(* IEC 61131-3 sources: elnaProjects/ElpcLogic/PomarKc7Changed/FunctionBlocks (part 3) *)

(* ---- Распаковка команды ---- *)
_sunpackerCommand(command := StrSw.inCommand);
	cmd := _sunpackerCommand.cmd;
	source := _sunpackerCommand.source;

(* ---- Обработка команды ---- *)
IF cmd <> 0 AND lastCmd <> cmd and (((NOT StrSw.opcCommandsDisabled) AND source > 0) OR source = 0) then
	CASE BYTE_TO_INT(cmd) OF
	(*cmd_open*) 1 :
			IF  StrSw.ISVALIDREF_cmdOn THEN StrSw.CmdOn := TRUE;
				IF StrSw.ISVALIDREF_cmdOff THEN StrSw.CmdOff := FALSE; END_IF;
			ELSIF  StrSw.ISVALIDREF_cmdOff THEN StrSw.CmdOff := FALSE;  END_IF;
			errorCMDTimer(IN := false);
			_commandErrorTimer := true;
			StrSw.lastCmdIsOn := true;
	(*cmd_close*) 2 :
			IF StrSw.ISVALIDREF_cmdOff THEN StrSw.CmdOff := TRUE;
				IF StrSw.ISVALIDREF_cmdOn THEN StrSw.CmdOn := FALSE; END_IF;
			ELSIF StrSw.ISVALIDREF_cmdOn THEN StrSw.CmdOn := FALSE; END_IF;
			errorCMDTimer(IN := false);
			_commandErrorTimer := true;
			StrSw.lastCmdIsOn := false;
	(*cmd_reset*) 3 :    IF StrSw.ISVALIDREF_statOn OR StrSw.ISVALIDREF_statOff THEN
			StrSw.CmdOn := FALSE;
			StrSw.CmdOff := FALSE;
                              lastCmd := 0;
			_commandErrorTimer := false;
			StrSw.lastCmdIsOn := false;
                               END_IF;
	END_CASE;
	source_for_Status := source;
	cmd_for_Status := cmd;
	command_error_for_Status := 0;
END_IF;
lastCmd := cmd;

errorCMDTimer(In := _commandErrorTimer, PT :=T#10s);

(* ---- алгоритм  для команды ВКЛючить ---- *)
IF (StrSw.onStatus = _statusDualInput.STATUS_ON) and (StrSw.lastCmdIsOn) then
	IF StrSw.ISVALIDREF_cmdOn AND StrSw.ISVALIDREF_cmdOff then  StrSw.cmdOn := false; END_IF;

	 errorCMDTimer(In := false);
	 _commandErrorTimer := false;
	 cmd_for_Status := 0;
	 source_for_Status := 0;
END_IF;

(* ---- off ---- *)
IF (StrSw.onStatus = _statusDualInput.STATUS_OFF) and (NOT StrSw.lastCmdIsOn) then
	IF StrSw.ISVALIDREF_cmdOn AND StrSw.ISVALIDREF_cmdOff then  StrSw.cmdOff := false; END_IF;

	 errorCMDTimer(In := false);
	 _commandErrorTimer := false;
	 cmd_for_Status := 0;
	 source_for_Status := 0;
END_IF;

(* ---- ошибка исполнения команды ---- *)
if errorCMDTimer.Q and (cmd_for_Status <> 0) then
	command_error_for_Status :=  cmd_for_Status;
	_commandErrorTimer := false;
	StrSw.CmdOn := false;
	StrSw.CmdOff := false;
	lastCmd := 0;
end_if;

(* ---- сброс ошибки команды ---- *)
StrSw.CommandFault := command_error_for_Status <> 0;
_errorReset(IN := command_error_for_Status <> 0, PT := T#5S);
IF _errorReset.Q THEN
	cmd_for_Status := 0;
	source_for_Status := 0;
	command_error_for_Status := 0;
END_IF;

outputsSets(in := (StrSw.ISVALIDREF_cmdOn and StrSw.cmdOn ) OR (StrSw.ISVALIDREF_cmdOff and StrSw.cmdOff), PT := T#2S);
	IF NOT outputsSets.Q THEN
		StrSw.BreakCmdOn := inBreakCmdOn._inversed AND inBreakCmdOn.reliability AND StrSw.ISVALIDREF_inBreakCmdOn;
		StrSw.BreakCmdOff := inBreakCmdOff._inversed AND inBreakCmdOff.reliability AND StrSw.ISVALIDREF_inBreakCmdOff;
	END_IF;

cmdOn := StrSw.cmdOn;
cmdOff:= StrSw.cmdOff;

(* ---- формирование зашифрованного статуса для АРМа ---- *)
StrSw.status := shl(BYTE_TO_DWORD(source_for_Status), 29)
		OR shl(BYTE_TO_DWORD(cmd_for_Status), 26)
		OR shl(BYTE_TO_DWORD(command_error_for_Status), 23)
		OR shl(bool_to_DWORD(StrSw.sdvig), 22)
		OR shl(bool_to_DWORD(StrSw.OpcCommandsDisabled), 21)
                    OR shl(BOOL_TO_DWORD(StrSw.offKNA), 17)
                    OR shl(bool_to_DWORD(StrSw.lastCmdIsOn), 14)
                    OR shl(BOOL_TO_DWORD(StrSw.BreakCmdOff), 13)
		OR shl(BOOL_TO_DWORD(StrSw.BreakCmdOn), 12)
                    OR shl(BYTE_TO_DWORD(StrSw.basketStatus), 8)
		OR shl(BOOL_TO_DWORD(StrSw.Distance), 6)
		OR shl(BOOL_TO_DWORD(StrSw.Local), 5)
		OR shl(BOOL_TO_DWORD(StrSw.Ns), 4)
                	OR shl(BOOL_TO_DWORD(StrSw.Accident ),3)
		OR BYTE_TO_DWORD(StrSw.onStatus);

(* ---- fb_SectionSwitch_Init.st ---- *)
FUNCTION_BLOCK fb_SectionSwitch_Init

VAR_INPUT
	data_Ini : BOOL; (*Флаг необходимости инициализации параметров.*)
	ISVALIDREF_statOn : BOOL;
	ISVALIDREF_statOff : BOOL;
	ISVALIDREF_cmdOn : BOOL;
	ISVALIDREF_cmdOff : BOOL;
	ISVALIDREF_inBreakCmdOn : BOOL;
	ISVALIDREF_inBreakCmdOff : BOOL;
	ISVALIDREF_basketRolledIn : BOOL;
	ISVALIDREF_basketRolledOut : BOOL;
	ISVALIDREF_basketTest : BOOL;
END_VAR

VAR_IN_OUT
	str_Sw : struct_SectionSwitch; (*Дескриптор AI-канала.*)
END_VAR

VAR_OUTPUT
	Init : BOOL          := FALSE; (*Флаг успешно выполненной инициализации.*)
END_VAR

(*****            Функциональный блок переинициализации структуры  МВ          *****)

 Init := FALSE;

    IF data_Ini THEN                            (* Параметрам требуется переинициализация. *)
        str_Sw.ISVALIDREF_statOn                := ISVALIDREF_statOn;
        str_Sw.ISVALIDREF_statOff               := ISVALIDREF_statOff;
        str_Sw.ISVALIDREF_cmdOn                 := ISVALIDREF_cmdOn;
        str_Sw.ISVALIDREF_cmdOff                := ISVALIDREF_cmdOff;
        str_Sw.ISVALIDREF_inBreakCmdOn          := ISVALIDREF_inBreakCmdOn;
        str_Sw.ISVALIDREF_inBreakCmdOff         := ISVALIDREF_inBreakCmdOff;
        str_Sw.ISVALIDREF_basketRolledIn        := ISVALIDREF_basketRolledIn;
        str_Sw.ISVALIDREF_basketRolledOut       := ISVALIDREF_basketRolledOut;
        str_Sw.ISVALIDREF_basketTest            := ISVALIDREF_basketTest;
        data_Ini:=FALSE;
        Init := TRUE;
    END_IF;
IF Init THEN
        ISVALIDREF_statOn:= FALSE;
        ISVALIDREF_statOff:= FALSE;
        ISVALIDREF_cmdOn:= FALSE;
        ISVALIDREF_cmdOff:= FALSE;
        ISVALIDREF_inBreakCmdOn:= FALSE;
        ISVALIDREF_inBreakCmdOff:= FALSE;
        ISVALIDREF_basketRolledIn:= FALSE;
        ISVALIDREF_basketRolledOut:= FALSE;
        ISVALIDREF_basketTest:= FALSE;
END_IF;

(* ---- fb_singleOutput.st ---- *)
FUNCTION_BLOCK fb_singleOutput

VAR_IN_OUT
	signal : BOOL;
	str_SO : struct_singleOutput;
END_VAR

VAR
	pulseTimer : TON;
	resetCmdTimer : TON;
	TON_Command : TON;
	source : BYTE;
	cmd : BYTE;
	lastCmd : BYTE;
	source_for_Status : BYTE;
	cmd_for_Status : BYTE;
	command_error_for_Status : BYTE;
	pulseTimerPriznak : BOOL;
	resetCmdTimerPriznak : BOOL;
	_sunpackerCommand : fb_sunpackerCommand;
END_VAR

str_SO.OpcCommandsDisabled := str_SO.inOpcCommandsDisabled;

(* ---- Если управление с ВУ заблокировано, то передаем команду из алгоритма ---- *)
IF str_SO.inOpcCommandsDisabled THEN
	str_SO.inCommand := str_SO.inCommand_Alg;
ELSE (* иначе передаем команду с АРМа*)
	str_SO.inCommand := str_SO.inCommand_ARM;
END_IF;

(*Распаковка команды*)
_sunpackerCommand(command := str_SO.inCommand);
	cmd := _sunpackerCommand.cmd;
	source := _sunpackerCommand.source;

(*Обработка команды*)
IF cmd <> 0 AND lastCmd <> cmd and (((NOT str_SO.OpcCommandsDisabled) AND source > 0) OR source = 0) then
	CASE BYTE_TO_INT(cmd) OF
	(*cmd_on*) 1 :
			str_SO.Q := TRUE;
			pulseTimer(IN := FALSE);
			pulseTimerPriznak := FALSE;
			resetCmdTimer(IN := FALSE);
			resetCmdTimerPriznak := TRUE;
	(*cmd_off*) 2 :
			str_SO.Q := FALSE;
			pulseTimer(IN := FALSE);
			pulseTimerPriznak := FALSE;
			resetCmdTimer(IN := FALSE);
			resetCmdTimerPriznak := TRUE;
	(*cmd_pulse*) 3 :
			str_SO.Q := TRUE;
                              pulseTimer(IN := FALSE);
                              pulseTimerPriznak := TRUE;
			resetCmdTimer(IN := FALSE);
                              resetCmdTimerPriznak := FALSE;
	END_CASE;
	source_for_Status := source;
	cmd_for_Status := cmd;
	command_error_for_Status := 0;
END_IF;
lastCmd := cmd;

pulseTimer(IN := pulseTimerPriznak, PT := str_SO.wait_time);
pulseTimer();
IF pulseTimer.Q THEN
	pulseTimer(IN := FALSE);
	pulseTimerPriznak := FALSE;

	str_SO.Q := FALSE;

	source_for_Status := 0;
	cmd_for_Status := 0;
	command_error_for_Status := 0;
END_IF;

resetCmdTimer(IN := resetCmdTimerPriznak, PT := T#10S);
resetCmdTimer();
IF resetCmdTimer.Q THEN
	resetCmdTimer(IN := FALSE);
	resetCmdTimerPriznak := FALSE;

	source_for_Status := 0;
	cmd_for_Status := 0;
	command_error_for_Status := 0;
END_IF;

signal:= str_SO.Q;

(*TON_Command(IN:= (inCommand <> 0) AND (source = 0), PT:= T#2S);*)
    (*IF TON_Command.Q THEN*)
        (*inCommand := 0;*)
    (*END_IF;*)
str_SO.status :=                           shl(BYTE_TO_DWORD(source_for_Status), 29)
				OR shl(BYTE_TO_DWORD(cmd_for_Status), 26)
				OR shl(BYTE_TO_DWORD(command_error_for_Status), 23)
				OR shl(BOOL_TO_DWORD(str_SO.OpcCommandsDisabled), 21)
				OR BOOL_TO_DWORD(str_SO.Q);

(* ---- fb_singleOutput_Init.st ---- *)
FUNCTION_BLOCK fb_singleOutput_Init

VAR_INPUT
	data_Ini : BOOL; (*Флаг необходимости инициализации параметров.*)
	inOpcCommandsDisabled : BOOL;
	wait_time : TIME;
END_VAR

VAR_IN_OUT
	str_SO : struct_singleOutput; (*Дескриптор AI-канала.*)
END_VAR

VAR_OUTPUT
	Init : BOOL          := FALSE; (*Флаг успешно выполненной инициализации.*)
END_VAR

(*****            Функциональный блок переинициализации структуры  singleOutput          *****)

Init := FALSE;

    IF data_Ini THEN                            (* Параметрам требуется переинициализация. *)
        str_SO.inOpcCommandsDisabled    := inOpcCommandsDisabled;
        str_SO.wait_time                := wait_time;

         data_Ini:=FALSE;
        Init := TRUE;
    END_IF;
 IF Init THEN
        inOpcCommandsDisabled := FALSE;
        wait_time := T#0S;
   END_IF;

(* ---- fb_singleSignal.st ---- *)
FUNCTION_BLOCK fb_singleSignal

VAR_INPUT
	signal : TYPE_ReliableBit;
END_VAR

VAR_IN_OUT
	str_SS : struct_singleSignal;
END_VAR

VAR
	TimerOn : TON;
	TimerOff : TOF;
END_VAR

str_SS.reliability:=signal.reliability;

IF NOT str_SS.inverse THEN
TimerOn(IN:=(signal.value AND str_SS.reliability AND NOT str_SS.Disabled_Sig), PT:=str_SS.DelayOn);
ELSE
TimerOn(IN:=(signal._inversed AND str_SS.reliability AND NOT str_SS.Disabled_Sig), PT:=str_SS.DelayOn);
END_IF;

TimerOff(IN:=TimerOn.Q, PT:=str_SS.DelayOff);

str_SS.Q:=TimerOff.Q;

str_SS.status:= SHL(BOOL_TO_DWORD(NOT str_SS.reliability), 15)
	OR BOOL_TO_DWORD(str_SS.Q);

(* ---- fb_singleSignal_Init.st ---- *)
FUNCTION_BLOCK fb_singleSignal_Init

VAR_INPUT
	data_Ini : BOOL; (*Флаг необходимости инициализации параметров.*)
	inverse : BOOL;
	DelayOn : TIME;
	DelayOff : TIME;
END_VAR

VAR_IN_OUT
	str_SS : struct_singleSignal; (*Дескриптор AI-канала.*)
END_VAR

VAR_OUTPUT
	Init : BOOL          := FALSE; (*Флаг успешно выполненной инициализации.*)
END_VAR

(*****            Функциональный блок переинициализации структуры  singleSignal          *****)
Init := FALSE;

    IF data_Ini THEN                            (* Параметрам требуется переинициализация. *)
        str_SS.inverse                := inverse;
        str_SS.DelayOn                := DelayOn;
        str_SS.DelayOff               := DelayOff;

        data_Ini:=FALSE;
        Init := TRUE;
    END_IF;
 IF Init THEN
        inverse := FALSE;
        DelayOn := T#0S;
        DelayOff:= T#0S;
 END_IF;

(* ---- fb_sunpackerCommand.st ---- *)
FUNCTION_BLOCK fb_sunpackerCommand

VAR_INPUT
	command : WORD;
END_VAR

VAR_OUTPUT
	source : BYTE;
	parametr : BYTE;
	cmd : BYTE;
END_VAR

cmd := WORD_TO_BYTE(command and 16#7);
parametr := WORD_TO_BYTE(SHR((command and 16#1FF8), 3));
source := WORD_TO_BYTE(SHR(command, 13));

(* ---- fb_Switch.st ---- *)
FUNCTION_BLOCK fb_Switch

VAR_INPUT
	statOn : BOOL;
	statOff : BOOL;
	statOn_reliability : BOOL;
	statOff_reliability : BOOL;
END_VAR

VAR_IN_OUT
	StrSw : struct_Switch;
END_VAR

VAR_INPUT
	inNs : TYPE_ReliableBit;
	inAccident : TYPE_ReliableBit;
	inAuto : TYPE_ReliableBit;
	inManual : TYPE_ReliableBit;
	inLocal : TYPE_ReliableBit;
	inDistance : TYPE_ReliableBit;
	inErrorPowerOff : TYPE_ReliableBit;
	inErrorBlock : TYPE_ReliableBit;
	inBreakCmdOn : TYPE_ReliableBit;
	inBreakCmdOff : TYPE_ReliableBit;
END_VAR

VAR
	onInit : BOOL          := FALSE;
	_statOn : BOOL;
	_statOff : BOOL;
	lastOnStatus : BYTE;
	cmd : BYTE;
	source : BYTE;
	lastCmd : BYTE;
	source_for_Status : BYTE;
	cmd_for_Status : BYTE;
	command_error_for_Status : BYTE;
	_sunpackerCommand : fb_sunpackerCommand;
	_statusDualInput : TYPE_statusDualInput;
	_commandDualInput : TYPE_commandDualInput;
	_commandErrorTimer : BOOL;
	resetErrorTimer : BOOL;
	getSdvig : BOOL;
	_changWithoutCommand : BOOL;
	errorCMDTimer : TON;
	sdvigReset : TON;
	_errorReset : TON;
	outputsSets : TOF;
END_VAR

VAR_IN_OUT
	cmdOn : BOOL;
	cmdOff : BOOL;
END_VAR

IF NOT onInit THEN
IF StrSw.ISVALIDREF_cmdOn XOR StrSw.ISVALIDREF_cmdOff THEN
	IF 	StrSw.ISVALIDREF_cmdOn THEN
		lastCmd:= 2; (*baseCmdOff*)
	ELSE
		lastCmd:= 1; (*baseCmdOn*)
	END_IF;
END_IF;
onInit:=TRUE;
END_IF;

(* ---- Если управление с ВУ заблокировано, то в ИМ передаем команду из алгоритма ---- *)
IF StrSw.inOpcCommandsDisabled THEN
	StrSw.inCommand := StrSw.inCommand_Alg;
ELSE (* иначе передаем команду с АРМа*)
	StrSw.inCommand := StrSw.inCommand_ARM;
END_IF;

(* ---- Формирование состояния механизма ---- *)

IF (StrSw.ISVALIDREF_statOn) OR (StrSw.ISVALIDREF_statOff) THEN
	IF (StrSw.ISVALIDREF_statOn) AND (StrSw.ISVALIDREF_statOff) THEN
	StrSw.reliability:= statOn_reliability AND statOff_reliability;
		_statOn  := statOn;
		_statOff := statOff;
	ELSIF (StrSw.ISVALIDREF_statOn) THEN
                     StrSw.reliability:= statOn_reliability;
		_statOn  := statOn;
		_statOff := NOT statOn;
	ELSIF (StrSw.ISVALIDREF_statOff) THEN
		 StrSw.reliability:= statOff_reliability;
		_statOn  := NOT statOff;
		_statOff :=statOff;
	END_IF;

	IF StrSw.reliability THEN
		IF _statOn AND NOT _statOff 		THEN 	StrSw.onStatus := _statusDualInput.STATUS_ON;
		ELSIF _statOff AND NOT _statOn 	THEN 	StrSw.onStatus := _statusDualInput.Status_OFF;
		ELSIF NOT _statOn AND NOT _statOff 	THEN 	StrSw.onStatus := _statusDualInput.STATUS_TRANSITIONAL;
		ELSE					StrSw.onStatus := _statusDualInput.STATUS_ERROR;
                    END_IF;

	ELSE
		StrSw.onStatus := _statusDualInput.STATUS_NOTDEFINED;

	END_IF;
ELSE
	CASE BYTE_TO_INT(lastCmd) OF
		(*baseCmdOn*) 1: StrSw.onStatus  := _statusDualInput.STATUS_ON;
		(*baseCmdOff*) 2: StrSw.onStatus  := _statusDualInput.STATUS_OFF;

	ELSE
		 StrSw.onStatus := _statusDualInput.STATUS_NOTDEFINED;

	END_CASE;
END_IF;

StrSw.Accident := inAccident.value AND inAccident.reliability;
StrSw.Ns := inNs.value AND inNs.reliability;
StrSw.Auto := inAuto.value AND inAuto.reliability;
StrSw.Manual := inManual.value AND inManual.reliability;
StrSw.Local := inLocal.value AND inLocal.reliability;
StrSw.Distance := inDistance.value AND inDistance.reliability;
StrSw.ErrorPowerOff := inErrorPowerOff.value AND inErrorPowerOff.reliability;
StrSw.ErrorBlock := inErrorBlock.value AND inErrorBlock.reliability;
StrSw.OpcCommandsDisabled := StrSw.inOpcCommandsDisabled;

(* ---- Формирование признака сдвига ---- *)
getSdvig := FALSE;
IF (StrSw.ISVALIDREF_cmdOn OR StrSw.ISVALIDREF_cmdOff) AND NOT StrSw.Local THEN
	IF NOT (StrSw.CmdOn OR StrSw.CmdOff) THEN
                     IF (lastOnStatus <> StrSw.onStatus AND
		(StrSw.onStatus <> _statusDualInput.STATUS_NOTDEFINED AND
                     StrSw.onStatus <> _statusDualInput.STATUS_ERROR)     AND
		(lastOnStatus <> _statusDualInput.STATUS_NOTDEFINED   AND
                     lastOnStatus <> _statusDualInput.STATUS_ERROR))
                    THEN
			getSdvig   := TRUE;
		END_IF;
	END_IF;
END_IF;

IF getSdvig THEN StrSw.sdvig:= TRUE; END_IF;

sdvigReset(IN:=StrSw.sdvig, PT:=T#15S);

IF sdvigReset.Q THEN StrSw.sdvig:=FALSE; END_IF;

lastOnStatus := StrSw.onStatus;

(* ---- Распаковка команды ---- *)
_sunpackerCommand(command := StrSw.inCommand);
	cmd := _sunpackerCommand.cmd;
	source := _sunpackerCommand.source;

(* ---- Обработка команды ---- *)
IF cmd <> 0 AND lastCmd <> cmd and (((NOT StrSw.opcCommandsDisabled) AND source > 0) OR source = 0) then
	CASE BYTE_TO_INT(cmd) OF
	(*cmd_open*) 1 :
			IF  StrSw.ISVALIDREF_cmdOn THEN StrSw.CmdOn := TRUE;
				IF StrSw.ISVALIDREF_cmdOff THEN StrSw.CmdOff := FALSE; END_IF;
			ELSIF  StrSw.ISVALIDREF_cmdOff THEN StrSw.CmdOff := FALSE;  END_IF;
                              lastCmd := cmd;
			errorCMDTimer(IN := false);
			_commandErrorTimer := true;
			StrSw.lastCmdIsOn := true;
	(*cmd_close*) 2 :
			IF StrSw.ISVALIDREF_cmdOff THEN StrSw.CmdOff := TRUE;
				IF StrSw.ISVALIDREF_cmdOn THEN StrSw.CmdOn := FALSE; END_IF;
			ELSIF StrSw.ISVALIDREF_cmdOn THEN StrSw.CmdOn := FALSE; END_IF;
                              lastCmd := cmd;
			errorCMDTimer(IN := false);
			_commandErrorTimer := true;
			StrSw.lastCmdIsOn := false;
	(*cmd_reset*) 3 :    IF StrSw.ISVALIDREF_statOn OR StrSw.ISVALIDREF_statOff THEN
			StrSw.CmdOn := FALSE;
			StrSw.CmdOff := FALSE;
                              lastCmd :=0;
			_commandErrorTimer := false;
			StrSw.lastCmdIsOn := false;
                               END_IF;
	END_CASE;
	source_for_Status := source;
	cmd_for_Status := cmd;
	command_error_for_Status := 0;
END_IF;

errorCMDTimer(In := _commandErrorTimer, PT :=T#10s);

(* ---- алгоритм  для команды ВКЛючить ---- *)
IF (StrSw.onStatus = _statusDualInput.STATUS_ON) and StrSw.lastCmdIsOn then
	IF StrSw.ISVALIDREF_cmdOn AND StrSw.ISVALIDREF_cmdOff then  StrSw.cmdOn := false; END_IF;

	 errorCMDTimer(In := false);
	 _commandErrorTimer := false;
	 cmd_for_Status := 0;
	 source_for_Status := 0;
END_IF;

(* ---- off ---- *)
IF (StrSw.onStatus = _statusDualInput.STATUS_OFF) and (NOT StrSw.lastCmdIsOn) then
	IF StrSw.ISVALIDREF_cmdOn AND StrSw.ISVALIDREF_cmdOff then  StrSw.cmdOff := false; END_IF;

	 errorCMDTimer(In := false);
	 _commandErrorTimer := false;
	 cmd_for_Status := 0;
	 source_for_Status := 0;
END_IF;

(* ---- ошибка исполнения команды ---- *)
if errorCMDTimer.Q and (cmd_for_Status <> 0) then
	command_error_for_Status :=  cmd_for_Status;
	_commandErrorTimer := false;
	StrSw.CmdOn := false;
	StrSw.CmdOff := false;
	lastCmd := 0;
end_if;

(* ---- сброс ошибки команды ---- *)
StrSw.CommandFault := command_error_for_Status <> 0;
_errorReset(IN := command_error_for_Status <> 0, PT := T#5S);
IF _errorReset.Q THEN
	cmd_for_Status := 0;
	source_for_Status := 0;
	command_error_for_Status := 0;
END_IF;

outputsSets(in := (StrSw.ISVALIDREF_cmdOn and StrSw.cmdOn ) OR (StrSw.ISVALIDREF_cmdOff and StrSw.cmdOff), PT := T#2S);
	IF NOT outputsSets.Q THEN
		StrSw.BreakCmdOn := inBreakCmdOn._inversed AND
                    inBreakCmdOn.reliability AND StrSw.ISVALIDREF_inBreakCmdOn;

		StrSw.BreakCmdOff := inBreakCmdOff._inversed
                    AND inBreakCmdOff.reliability AND StrSw.ISVALIDREF_inBreakCmdOff;
	END_IF;

cmdOn := StrSw.cmdOn;
cmdOff:= StrSw.cmdOff;

(* ---- формирование зашифрованного статуса для АРМа ---- *)
StrSw.status := shl(BYTE_TO_DWORD(source_for_Status), 29)
		OR shl(BYTE_TO_DWORD(cmd_for_Status), 26)
		OR shl(BYTE_TO_DWORD(command_error_for_Status), 23)
		OR shl(bool_to_DWORD(StrSw.sdvig), 22)
		OR shl(bool_to_DWORD(StrSw.OpcCommandsDisabled), 21)
                    OR shl(bool_to_DWORD(StrSw.lastCmdIsOn), 14)
                    OR shl(BOOL_TO_DWORD(StrSw.BreakCmdOff), 13)
		OR shl(BOOL_TO_DWORD(StrSw.BreakCmdOn), 12)
		OR shl(BOOL_TO_DWORD(StrSw.ErrorBlock), 11)
		OR shl(BOOL_TO_DWORD(StrSw.ErrorPowerOff), 10)
		OR shl(BOOL_TO_DWORD(StrSw.Manual), 8)
		OR shl(BOOL_TO_DWORD(StrSw.Auto), 7)
		OR shl(BOOL_TO_DWORD(StrSw.Distance), 6)
		OR shl(BOOL_TO_DWORD(StrSw.Local), 5)
		OR shl(BOOL_TO_DWORD(StrSw.Ns), 4)
                	OR shl(BOOL_TO_DWORD(StrSw.Accident ),3)
		OR BYTE_TO_DWORD(StrSw.onStatus);

(* ---- fb_Switch_Init.st ---- *)
FUNCTION_BLOCK fb_Switch_Init

VAR_INPUT
	data_Ini : BOOL; (*Флаг необходимости инициализации параметров.*)
	ISVALIDREF_statOn : BOOL;
	ISVALIDREF_statOff : BOOL;
	ISVALIDREF_cmdOn : BOOL;
	ISVALIDREF_cmdOff : BOOL;
	ISVALIDREF_inBreakCmdOn : BOOL;
	ISVALIDREF_inBreakCmdOff : BOOL;
END_VAR

VAR_IN_OUT
	str_Sw : struct_Switch;
END_VAR

VAR_OUTPUT
	Init : BOOL          := FALSE; (*Флаг успешно выполненной инициализации.*)
END_VAR

(*****            Функциональный блок переинициализации структуры  Switch          *****)

 Init := FALSE;

    IF data_Ini THEN                            (* Параметрам требуется переинициализация. *)
        str_Sw.ISVALIDREF_statOn                := ISVALIDREF_statOn;
        str_Sw.ISVALIDREF_statOff               := ISVALIDREF_statOff;
        str_Sw.ISVALIDREF_cmdOn                 := ISVALIDREF_cmdOn;
        str_Sw.ISVALIDREF_cmdOff                := ISVALIDREF_cmdOff;
        str_Sw.ISVALIDREF_inBreakCmdOn          := ISVALIDREF_inBreakCmdOn;
        str_Sw.ISVALIDREF_inBreakCmdOff         := ISVALIDREF_inBreakCmdOff;
        data_Ini:=FALSE;
        Init := TRUE;
    END_IF;
IF Init THEN
        ISVALIDREF_statOn:= FALSE;
        ISVALIDREF_statOff:= FALSE;
        ISVALIDREF_cmdOn:= FALSE;
        ISVALIDREF_cmdOff:= FALSE;
        ISVALIDREF_inBreakCmdOn:= FALSE;
        ISVALIDREF_inBreakCmdOff:= FALSE;
END_IF;

(* ---- fb_TableValue_Max.st ---- *)
FUNCTION_BLOCK fb_TableValue_Max

VAR_INPUT
	parametr : REAL;
END_VAR

VAR
	_table : ARRAY [0..8] OF TYPE_TableRec;
END_VAR

VAR_INPUT
	inverse : BOOL          := FALSE;
END_VAR

VAR_IN_OUT
	actualValue : REAL;
END_VAR

VAR
	indexLess : INT          := -1;
	indexMore : INT          := -1;
	Vali : REAL;
	i : INT;
	moreDistance : REAL;
	lessDistance : REAL;
	onInit : BOOL;
	_prevParam : REAL          := 50.0;
END_VAR

VAR CONSTANT
	maxTableLength : INT          := 9;
END_VAR

IF NOT onInit THEN
_table[0].x:=-35.0;  _table[0].y:=320.0;
_table[1].x:=-25.0;  _table[1].y:=315.0;
_table[2].x:=-15.0;  _table[2].y:=310.0;
_table[3].x:= -5.0;  _table[3].y:=305.0;
_table[4].x:=  0.0;  _table[4].y:=300.0;
_table[5].x:=  5.0;  _table[5].y:=295.0;
_table[6].x:= 15.0;  _table[6].y:=290.0;
_table[7].x:= 25.0;  _table[7].y:=285.0;
_table[8].x:= 35.0;  _table[8].y:=280.0;

onInit:=TRUE;
END_IF;

IF parametr <> _prevParam THEN
indexLess:=-1;
indexMore:=-1;
lessDistance:=0.0;
moreDistance:=0.0;
FOR i:=0 TO maxTableLength-1 DO
	IF NOT inverse THEN
		Vali:=_table[i].x;
	ELSE
		Vali:=_table[i].y;
	END_IF;

	IF (Vali=parametr) THEN
		indexLess:=i;
		indexMore:=i;
	ELSIF ((Vali<parametr) AND ((lessDistance>parametr-Vali) OR (indexLess<0))) THEN
		indexLess:=i;
		lessDistance:=parametr-Vali;
	ELSIF ((Vali>parametr) AND ((moreDistance>Vali-parametr) OR (indexMore<0))) THEN
		indexMore:=i;
		moreDistance:=parametr-Vali;
	END_IF;
END_FOR;
(*
IF indexLess<0 THEN
	indexLess:=indexMore;
END_IF;

IF indexMore<0 THEN
	indexMore:=indexLess;
END_IF;
*)
  IF (_table[indexMore].x<>_table[indexLess].x) THEN
  actualValue:=_table[indexLess].y+((_table[indexMore].y-_table[indexLess].y)/(_table[indexMore].x-_table[indexLess].x))*(parametr-_table[indexLess].x);
  ELSE
  actualValue:=_table[indexLess].y;
  END_IF;
   _prevParam:= parametr;
END_IF;

(* ---- fb_TableValue_Min.st ---- *)
FUNCTION_BLOCK fb_TableValue_Min

VAR_INPUT
	parametr : REAL;
END_VAR

VAR
	_table : ARRAY [0..8] OF TYPE_TableRec;
END_VAR

VAR_INPUT
	inverse : BOOL          := FALSE;
END_VAR

VAR_IN_OUT
	actualValue : REAL;
END_VAR

VAR
	indexLess : INT          := -1;
	indexMore : INT          := -1;
	Vali : REAL;
	i : INT;
	moreDistance : REAL;
	lessDistance : REAL;
	onInit : BOOL;
	_prevParam : REAL          := 50.0;
END_VAR

VAR CONSTANT
	maxTableLength : INT          := 9;
END_VAR

IF NOT onInit THEN
_table[0].x:=-35.0;  _table[0].y:=130.0;
_table[1].x:=-25.0;  _table[1].y:=124.0;
_table[2].x:=-15.0;  _table[2].y:=118.0;
_table[3].x:= -5.0;  _table[3].y:=112.0;
_table[4].x:=  0.0;  _table[4].y:=108.0;
_table[5].x:=  5.0;  _table[5].y:=106.0;
_table[6].x:= 15.0;  _table[6].y:=104.0;
_table[7].x:= 25.0;  _table[7].y:=102.0;
_table[8].x:= 35.0;  _table[8].y:= 97.0;

onInit:=TRUE;
END_IF;

IF parametr <> _prevParam THEN
indexLess:=-1;
indexMore:=-1;
lessDistance:=0.0;
moreDistance:=0.0;
FOR i:=0 TO maxTableLength-1 DO
	IF NOT inverse THEN
		Vali:=_table[i].x;
	ELSE
		Vali:=_table[i].y;
	END_IF;

	IF (Vali=parametr) THEN
		indexLess:=i;
		indexMore:=i;
	ELSIF ((Vali<parametr) AND ((lessDistance>parametr-Vali) OR (indexLess<0))) THEN
		indexLess:=i;
		lessDistance:=parametr-Vali;
	ELSIF ((Vali>parametr) AND ((moreDistance>Vali-parametr) OR (indexMore<0))) THEN
		indexMore:=i;
		moreDistance:=parametr-Vali;
	END_IF;
END_FOR;
(*
IF indexLess<0 THEN
	indexLess:=indexMore;
END_IF;

IF indexMore<0 THEN
	indexMore:=indexLess;
END_IF;
*)
  IF (_table[indexMore].x<>_table[indexLess].x) THEN
  actualValue:=_table[indexLess].y+((_table[indexMore].y-_table[indexLess].y)/(_table[indexMore].x-_table[indexLess].x))*(parametr-_table[indexLess].x);
  ELSE
  actualValue:=_table[indexLess].y;
  END_IF;
   _prevParam:= parametr;
END_IF;

(* ---- fb_Timings.st ---- *)
FUNCTION_BLOCK fb_Timings

VAR_EXTERNAL CONSTANT
	req_Cycle : REAL;
END_VAR

VAR_EXTERNAL
	gF_T_100mSec : BOOL;
	gT_1Sec : BOOL;
	gF_T_1Sec : BOOL;
	gT_1Min : BOOL;
	gR_T_1Min : BOOL;
	gF_T_1Min : BOOL;
	del_T : REAL;
	cur_Cycle : REAL;
END_VAR

VAR
	Tmr_100_ms : REAL; (*Таймер меток времени 100 мс .*)
END_VAR

VAR_EXTERNAL
	T_1SEC : REAL;
END_VAR

VAR
	Tmr_1_s : REAL; (*Таймер меток времени 1 с .*)
	Tmr_1_min : REAL; (*Таймер меток времени 1 мин .*)
END_VAR

(* Обработка времени. *)
Tmr_100_ms := Tmr_100_ms + cur_Cycle;
gF_T_100mSec := FALSE;
IF Tmr_100_ms >= 0.1 THEN Tmr_100_ms := 0.0; gF_T_100mSec := TRUE; END_IF;

Tmr_1_s := Tmr_1_s + cur_Cycle;
gF_T_1Sec := FALSE;
IF Tmr_1_s >= 1.0 THEN Tmr_1_s := 0.0; gF_T_1Sec := TRUE; END_IF;

T_1SEC := T_1SEC + cur_Cycle;
gT_1Sec := FALSE;
IF T_1SEC >= 2.0 THEN T_1SEC := 0.0;
  ELSIF T_1SEC >= 1.0 THEN gT_1Sec := TRUE; END_IF;

IF Tmr_1_min > 60.0 THEN
    Tmr_1_min := 0.0; gF_T_1Min := gT_1Min; gT_1Min := NOT gT_1Min; gR_T_1Min := gT_1Min;
  ELSE
    Tmr_1_min := Tmr_1_min + cur_Cycle; gR_T_1Min := FALSE; gF_T_1Min := FALSE;
END_IF;
del_T:= cur_Cycle;

(* ---- fb_vibegPNSAlg.st ---- *)
FUNCTION_BLOCK fb_vibegPNSAlg

VAR_IN_OUT
	StrAlg : struct_Alg;
END_VAR

VAR
	autoPnsOff : struct_PhaseAlgoritm;
	waitVibeg : struct_PhaseAlgoritm;
	pnsOff : struct_PhaseAlgoritm;
	vibegEnd : struct_PhaseAlgoritm;
END_VAR

VAR_IN_OUT
	algContinue : struct_Question;
END_VAR

VAR
	fb_autoPnsOff : fb_ph_algoritm;
	fb_waitVibeg : fb_ph_Timer;
	fb_algContinue : fb_Question;
	fb_pnsOff : fb_ph_Switch;
	fb_vibegEnd : fb_ph_CustomPhase;
	_sunpackerCommand : fb_sunpackerCommand;
	_statusAi : TYPE_StatusAi;
	_Answers : TYPE_Answers;
	_statusDualInput : TYPE_statusDualInput;
	_DualStateImAction : TYPE_DualStateImAction;
	_PhaseAlgoritmAction : TYPE_PhaseAlgoritmAction;
	source : BYTE;
	cmd : BYTE;
	lastCmd : BYTE;
	source_for_Status : BYTE;
	cmd_for_Status : BYTE;
	command_error_for_Status : BYTE;
	resetCmdTimer : TON;
	resetCmdTimerPriznak : BOOL;
	onInit : BOOL;
	waitReset : TON;
END_VAR

VAR_EXTERNAL
	IM : ImConfig;
	algoritms : AlgoritmsConfig;
	ai : AiConfig;
	protections : ProtectionsConfig;
	AlgTimers : struct_AlgTimers;
END_VAR

IF NOT onInit THEN
 fb_autoPnsOff(phaseNumber:=0, act:=_reset, waitCompletion:=FALSE);
  fb_waitVibeg(phaseNumber:=1, delay:=T#300S);
     algContinue.AnswerVariants:=_Answers.ANS_YES;
     fb_pnsOff(phaseNumber:=2, act:=_off);
   fb_vibegEnd(phaseNumber:=14);
onInit:=TRUE;
END_IF;

 fb_autoPnsOff(StrPh:=autoPnsOff, alg:=algoritms.autoPns);
  fb_waitVibeg(StrPh:=waitVibeg, timer:=AlgTimers.vibegPNS_Timer);
fb_algContinue(StrQ:=algContinue);
     fb_pnsOff(StrPh:=pnsOff, Im:=IM.pns);
   fb_vibegEnd(StrPh:=vibegEnd);

IF StrAlg.isRuning THEN

StrAlg.hasError := autoPnsOff.error OR pnsOff.error;

    IF IM.pns.onStatus = _statusDualInput.STATUS_ON AND NOT vibegEnd.top THEN

	runPhase(vibegEnd);
          runPhase(waitVibeg);
          askQuestion(algContinue);

    END_IF;

    IF waitVibeg.top OR (algContinue.answer = _Answers.ANS_YES) THEN
	vibegEnd.top:=TRUE;
	resetPhase(waitVibeg);
          resetQuestion(algContinue);

          resetAiProtection(protections.Os_sdvig_nagnetatelja_minus);
          (*resetDiProtection(protections.Vibro_skorost_OP_shesterni_RED_T6);*)

	(*IM.SingleSignals.P_oil_low.Disabled_Sig:=TRUE;*)
	ai.Pmasla_posle_GNS.Disabled_LA:=TRUE;
          ai.Pmasla_posle_GNS.Disabled_LW:=TRUE;
          ai.Pmasla_posle_NU.Disabled_LW:=TRUE;
	runPhase(pnsOff);
    END_IF;

    StrAlg.isEnded:=pnsOff.top;

END_IF;

StrAlg.CanRun := StrAlg.inCanRun;
StrAlg.OpcCommandsDisabled := StrAlg.inOpcCommandsDisabled;

(* ---- Если управление с ВУ заблокировано, то  передаем команду из алгоритма ---- *)
IF StrAlg.inOpcCommandsDisabled THEN
	StrAlg.inCommand := StrAlg.inCommand_Alg;
ELSE (* иначе передаем команду с АРМа*)
	StrAlg.inCommand := StrAlg.inCommand_ARM;
END_IF;

_sunpackerCommand(command := StrAlg.inCommand);
	source := _sunpackerCommand.source;
	cmd := _sunpackerCommand.cmd;

IF cmd <> 0 AND lastCmd <> cmd AND (((NOT StrAlg.opcCommandsDisabled) AND source > 0) OR source = 0) then
	CASE BYTE_TO_INT(cmd) OF
		(*cmdRun*) 1: 	IF (StrAlg.CanRun) THEN
					StrAlg.isRuning := TRUE;
					StrAlg.isEnded := FALSE;
					StrAlg.hasError := FALSE;
					(*****************       OnRun       *****************)
                                                  runPhase(autoPnsOff);

					cmd_for_Status := cmd;
					source_for_Status := source;
					command_error_for_Status := 0;
				ELSE
					StrAlg.isRuning := FALSE;
					StrAlg.isEnded := FALSE;
					StrAlg.hasError 	:= FALSE;

					cmd_for_Status := 0;
					source_for_Status := source;
					command_error_for_Status := cmd;
				END_IF;
		(*cmdReset*) 2: 	StrAlg.isRuning := FALSE;
				StrAlg.isEnded := FALSE;
				StrAlg.hasError 	:= FALSE;

                                         (*****************       OnReset       *****************)
                                       waitReset(IN:=FALSE);
                                       resetPhase(autoPnsOff);
                                       resetPhase(waitVibeg);
                                       resetPhase(vibegEnd);
                                       resetPhase(pnsOff);
                                       resetQuestion(algContinue);

				cmd_for_Status := cmd;
				source_for_Status := source;
				command_error_for_Status := 0;
	END_CASE;
	resetCmdTimer(IN := false);
	resetCmdTimerPriznak := TRUE;
END_IF;
lastCmd := cmd;

resetCmdTimer(IN := resetCmdTimerPriznak, PT := T#5S);
IF resetCmdTimer.Q THEN
	resetCmdTimerPriznak := FALSE;
	source_for_Status := 0;
	cmd_for_Status := 0;
	command_error_for_Status := 0;
END_IF;

StrAlg.Start:= autoPnsOff.startStatus
            OR waitVibeg.startStatus
            OR pnsOff.startStatus
            OR vibegEnd.startStatus;

StrAlg.Error:= autoPnsOff.errorStatus
            OR waitVibeg.errorStatus
            OR pnsOff.errorStatus
            OR vibegEnd.errorStatus;

StrAlg.Top:=   autoPnsOff.topStatus
            OR waitVibeg.topStatus
            OR pnsOff.topStatus
            OR vibegEnd.topStatus;

(*TODO: TYPE PROGRAM CODE HERE*)
StrAlg.status :=  SHL(BYTE_TO_DWORD(source_for_Status), 29)
			OR SHL(BYTE_TO_DWORD(cmd_for_Status), 26)
			OR SHL(BYTE_TO_DWORD(command_error_for_Status), 23)
			OR SHL(BOOL_TO_DWORD(StrAlg.OpcCommandsDisabled ), 21)
			OR SHL(BOOL_TO_DWORD(StrAlg.hasError),4)
			OR SHL(BOOL_TO_DWORD(StrAlg.CanRun),2)
			OR SHL(BOOL_TO_DWORD(StrAlg.isEnded),1)
			OR BOOL_TO_DWORD(StrAlg.isRuning);

(* ---- fb_ZapasAlg.st ---- *)
FUNCTION_BLOCK fb_ZapasAlg

VAR_INPUT
	Q_actual : struct_AI;
END_VAR

VAR_IN_OUT
	StrAi : struct_AI;
END_VAR

VAR_INPUT
	Q_min : LREAL;
	Q_max : LREAL;
END_VAR

VAR
	_statusAi : TYPE_StatusAi;
END_VAR

IF (Q_actual.interval < _statusAi.normal) THEN
	StrAi.interval := _statusAi.NOTRELIABLE;
          strAI.status := 	SHL(BOOL_TO_DWORD(strAI.OpcCommandsDisabled ), 21)
		OR BYTE_TO_DWORD(strAI.interval);
	RETURN;
END_IF;

IF (Q_actual.value <10.0) THEN
	StrAi.interval := _statusAi.normal;
	StrAi.value:= 100.0;
          strAI.status := 	SHL(BOOL_TO_DWORD(strAI.OpcCommandsDisabled ), 21)
		OR BYTE_TO_DWORD(strAI.interval);
	RETURN;
END_IF;

strAI.opcCommandsDisabled := strAI.inopcCommandsDisabled ;
StrAi.interval:= _statusAi.normal;

StrAi.value:= ((Q_actual.value - Q_min)/(Q_max-Q_min))*100.0;

strAI.status := 	SHL(BOOL_TO_DWORD(strAI.OpcCommandsDisabled ), 21) (* Управление в ВУ заблокировано *)
		OR BYTE_TO_DWORD(strAI.interval);	              (* интервал *)

(* ---- fillingAlg.st ---- *)
FUNCTION_BLOCK fillingAlg

VAR_IN_OUT
	StrAlg : struct_Alg;
END_VAR

VAR
	BreakPuskTimer : struct_PhaseAlgoritm;
	kran3bOpen : struct_PhaseAlgoritm;
	kran4Open : struct_PhaseAlgoritm;
	waitAfterKran4 : struct_PhaseAlgoritm;
	kran5Close : struct_PhaseAlgoritm;
	didPKran1 : struct_PhaseAlgoritm;
	kran1Open : struct_PhaseAlgoritm;
	kran2Open : struct_PhaseAlgoritm;
	kran3bClose : struct_PhaseAlgoritm;
	kran4Close : struct_PhaseAlgoritm;
	RunProtection_kr1 : struct_PhaseAlgoritm;
	RunProtection_kr2 : struct_PhaseAlgoritm;
	waitAfterKran5 : struct_PhaseAlgoritm;
	testUnsuccessfulFilling : struct_PhaseAlgoritm;
	fb_BreakPuskTimer : fb_ph_Timer;
	fb_kran3bOpen : fb_ph_Kran;
	fb_kran4Open : fb_ph_Kran;
	fb_waitAfterKran4 : fb_ph_Timer;
	fb_kran5Close : fb_ph_Kran;
	fb_didPKran1 : fb_ph_CustomPhase;
	fb_kran1Open : fb_ph_Kran;
	fb_kran2Open : fb_ph_Kran;
	fb_kran3bClose : fb_ph_Kran;
	fb_kran4Close : fb_ph_Kran;
	fb_RunProtection_kr1 : fb_ph_DIprotection;
	fb_RunProtection_kr2 : fb_ph_DIprotection;
	fb_waitAfterKran5 : fb_ph_Timer;
	fb_testUnsuccessfulFilling : fb_ph_CustomPhase;
	_sunpackerCommand : fb_sunpackerCommand;
	_DualStateImAction : TYPE_DualStateImAction;
	_PhaseAlgoritmAction : TYPE_PhaseAlgoritmAction;
	source : BYTE;
	cmd : BYTE;
	lastCmd : BYTE;
	source_for_Status : BYTE;
	cmd_for_Status : BYTE;
	command_error_for_Status : BYTE;
	resetCmdTimer : TON;
	resetCmdTimerPriznak : BOOL;
	onInit : BOOL;
	waitReset : TON;
END_VAR

VAR_EXTERNAL
	IM : ImConfig;
	ai : AiConfig;
	protections : ProtectionsConfig;
	AlgTimers : struct_AlgTimers;
	algoritms : AlgoritmsConfig;
END_VAR

IF NOT onInit THEN

         fb_BreakPuskTimer(phaseNumber:=0, delay:=T#240S);
             fb_kran3bOpen(phaseNumber:=1, act:=_on);
              fb_kran4Open(phaseNumber:=2, act:=_on);
         fb_waitAfterKran4(phaseNumber:=3, delay:=T#10S);
             fb_kran5Close(phaseNumber:=4, act:=_off);
              fb_didPKran1(phaseNumber:=5);
              fb_kran1Open(phaseNumber:=7, act:=_on);
              fb_kran2Open(phaseNumber:=8, act:=_on);
            fb_kran3bClose(phaseNumber:=9, act:=_off);
             fb_kran4Close(phaseNumber:=10, act:=_off);
      fb_RunProtection_kr1(phaseNumber:=11, act:=_run);
      fb_RunProtection_kr2(phaseNumber:=12, act:=_run);
         fb_waitAfterKran5(phaseNumber:=13, delay:=T#60S);
fb_testUnsuccessfulFilling(phaseNumber:=17);

onInit:=TRUE;
END_IF;

         fb_BreakPuskTimer(StrPh:=BreakPuskTimer, timer:=AlgTimers.filling_BreakPuskTimer);
             fb_kran3bOpen(StrPh:=kran3bOpen, Im:=Im.kran3b);
              fb_kran4Open(StrPh:=kran4Open, Im:=Im.kran4);
         fb_waitAfterKran4(StrPh:=waitAfterKran4, timer:=AlgTimers.filling_waitAfterKran4);
             fb_kran5Close(StrPh:=kran5Close, Im:=Im.kran5);
              fb_didPKran1(StrPh:=didPKran1);
              fb_kran1Open(StrPh:=kran1Open, Im:=Im.kran1);
              fb_kran2Open(StrPh:=kran2Open, Im:=Im.kran2);
            fb_kran3bClose(StrPh:=kran3bClose, Im:=Im.kran3b);
             fb_kran4Close(StrPh:=kran4Close, Im:=Im.kran4);
      fb_RunProtection_kr1(StrPh:=RunProtection_kr1 , StrDiP:=protections.Reg_vozb_off);
      fb_RunProtection_kr2(StrPh:=RunProtection_kr2 , StrDiP:=protections.Fail_chastotnii_pusk);
         fb_waitAfterKran5(StrPh:=waitAfterKran5, timer:=AlgTimers.filling_waitAfterKran5);
fb_testUnsuccessfulFilling(StrPh:=testUnsuccessfulFilling);

StrAlg.CanRun := StrAlg.inCanRun;
StrAlg.OpcCommandsDisabled := StrAlg.inOpcCommandsDisabled;

IF StrAlg.isRuning THEN

    StrAlg.hasError := kran3bOpen.error OR kran4Open.error OR kran5Close.error OR kran5Close.error
    OR kran1Open.error OR kran2Open.error OR kran3bClose.error OR kran4Close.error OR testUnsuccessfulFilling.error;

    IF kran4Open.top THEN
        runPhase(waitAfterKran4);
    END_IF;

    IF waitAfterKran4.top THEN
        runPhase(kran5Close);
    END_IF;

    IF kran3bOpen.top AND kran5Close.top THEN
       runPhase(waitAfterKran5);
       runPhase(didPKran1);
    END_IF;

    (*IF didPKran1.start AND NOT didPKran1.top THEN
    didPKran1.top:= im.singleSignals.dP_gazgaz_Kran1.Q;
    END_IF;*)

    IF waitAfterKran5.top AND didPKran1.top THEN
          runPhase(kran1Open);
	runPhase(kran2Open);
    END_IF;

    IF kran1Open.top AND kran2Open.top THEN
          runPhase(kran4Close);
	runPhase(kran3bClose);
    END_IF;

    IF kran4Close.top AND kran3bClose.top THEN

          runPhase(RunProtection_kr1);
          runPhase(RunProtection_kr2);

          (*runAiProtection(protections.Pgaza_na_vhode_nagnetatelia);
          runAiProtection(protections.Pgaza_na_vhode_nagnetatelia);
          runAiProtection(protections.Pgaza_na_vyhode_nagnetatelia);
          runAiProtection(protections.dPmaslo_gaz);
          runAiProtection(protections.Pmaslo_sm_nizkoe);
          runAiProtection(protections.Pmaslo_sm_vysokoe);*)

    END_IF;

    IF BreakPuskTimer.top AND NOT (RunProtection_kr1.top AND RunProtection_kr2.top ) THEN
	testUnsuccessfulFilling.error:=TRUE;
    END_IF;

    IF RunProtection_kr1.top AND RunProtection_kr2.top THEN
          resetPhase(BreakPuskTimer);
	waitReset(IN:=TRUE, PT:= T#2S);
    END_IF;

    IF waitReset.Q AND NOT (algoritms.Apusk.isRuning OR algoritms.SemiAutoPusk.isRuning) THEN
	resetIfRunning(StrAlg);
    END_IF;

    StrAlg.isEnded:= RunProtection_kr1.top AND RunProtection_kr2.top;
END_IF;

StrAlg.CanRun := StrAlg.inCanRun;
StrAlg.OpcCommandsDisabled := StrAlg.inOpcCommandsDisabled;

(* ---- Если управление с ВУ заблокировано, то  передаем команду из алгоритма ---- *)
IF StrAlg.inOpcCommandsDisabled THEN
	StrAlg.inCommand := StrAlg.inCommand_Alg;
ELSE (* иначе передаем команду с АРМа*)
	StrAlg.inCommand := StrAlg.inCommand_ARM;
END_IF;

_sunpackerCommand(command := StrAlg.inCommand);
	source := _sunpackerCommand.source;
	cmd := _sunpackerCommand.cmd;

IF cmd <> 0 AND lastCmd <> cmd AND (((NOT StrAlg.opcCommandsDisabled) AND source > 0) OR source = 0) then
	CASE BYTE_TO_INT(cmd) OF
		(*cmdRun*) 1: 	IF (StrAlg.CanRun) THEN
					StrAlg.isRuning := TRUE;
					StrAlg.isEnded := FALSE;
					StrAlg.hasError := FALSE;
					(*****************       OnRun       *****************)

                                                  runPhase(kran3bOpen);
                                                  runPhase(kran4Open);
                                                  runPhase(BreakPuskTimer);
                                                  runPhase(testUnsuccessfulFilling);

					cmd_for_Status := cmd;
					source_for_Status := source;
					command_error_for_Status := 0;
				ELSE
					StrAlg.isRuning := FALSE;
					StrAlg.isEnded := FALSE;
					StrAlg.hasError 	:= FALSE;

					cmd_for_Status := 0;
					source_for_Status := source;
					command_error_for_Status := cmd;
				END_IF;
		(*cmdReset*) 2: 	StrAlg.isRuning := FALSE;
				StrAlg.isEnded := FALSE;
				StrAlg.hasError 	:= FALSE;

                                         (*****************       OnReset       *****************)
                                        StrAlg.inCanRun:=FALSE;
                                        waitReset(IN:=FALSE);

                                        resetPhase(BreakPuskTimer);
                                        resetPhase(kran3bOpen);
                                        resetPhase(kran4Open);
                                        resetPhase(waitAfterKran4);
                                        resetPhase(kran5Close);
                                        resetPhase(didPKran1);
                                        resetPhase(kran1Open);
                                        resetPhase(kran2Open);
                                        resetPhase(kran3bClose);
                                        resetPhase(kran4Close);
	                              resetPhase(RunProtection_kr1);
                                        resetPhase(RunProtection_kr2);
                                        resetPhase(waitAfterKran5);
                                        resetPhase(testUnsuccessfulFilling);

				cmd_for_Status := cmd;
				source_for_Status := source;
				command_error_for_Status := 0;
	END_CASE;
	resetCmdTimer(IN := false);
	resetCmdTimerPriznak := TRUE;
END_IF;
lastCmd := cmd;

resetCmdTimer(IN := resetCmdTimerPriznak, PT := T#5S);
IF resetCmdTimer.Q THEN
	resetCmdTimerPriznak := FALSE;
	source_for_Status := 0;
	cmd_for_Status := 0;
	command_error_for_Status := 0;
END_IF;

StrAlg.Start:= BreakPuskTimer.startStatus
            OR kran3bOpen.startStatus
            OR kran4Open.startStatus
            OR waitAfterKran4.startStatus
            OR kran5Close.startStatus
            OR didPKran1.startStatus
            OR kran1Open.startStatus
            OR kran2Open.startStatus
            OR kran3bClose.startStatus
            OR kran4Close.startStatus
            OR RunProtection_kr1.startStatus
            OR RunProtection_kr2.startStatus
            OR waitAfterKran5.startStatus
            OR testUnsuccessfulFilling.startStatus;

StrAlg.Error:= BreakPuskTimer.errorStatus
            OR kran3bOpen.errorStatus
            OR kran4Open.errorStatus
            OR waitAfterKran4.errorStatus
            OR kran5Close.errorStatus
            OR didPKran1.errorStatus
            OR kran1Open.errorStatus
            OR kran2Open.errorStatus
            OR kran3bClose.errorStatus
            OR kran4Close.errorStatus
            OR RunProtection_kr1.errorStatus
            OR RunProtection_kr2.errorStatus
            OR waitAfterKran5.errorStatus
            OR testUnsuccessfulFilling.errorStatus;

StrAlg.Top:=   BreakPuskTimer.topStatus
            OR kran3bOpen.topStatus
            OR kran4Open.topStatus
            OR waitAfterKran4.topStatus
            OR kran5Close.topStatus
            OR didPKran1.topStatus
            OR kran1Open.topStatus
            OR kran2Open.topStatus
            OR kran3bClose.topStatus
            OR kran4Close.topStatus
            OR RunProtection_kr1.topStatus
            OR RunProtection_kr2.topStatus
            OR waitAfterKran5.topStatus
            OR testUnsuccessfulFilling.topStatus;

(*TODO: TYPE PROGRAM CODE HERE*)
StrAlg.status :=  SHL(BYTE_TO_DWORD(source_for_Status), 29)
			OR SHL(BYTE_TO_DWORD(cmd_for_Status), 26)
			OR SHL(BYTE_TO_DWORD(command_error_for_Status), 23)
			OR SHL(BOOL_TO_DWORD(StrAlg.OpcCommandsDisabled ), 21)
			OR SHL(BOOL_TO_DWORD(StrAlg.hasError),4)
			OR SHL(BOOL_TO_DWORD(StrAlg.CanRun),2)
			OR SHL(BOOL_TO_DWORD(StrAlg.isEnded),1)
			OR BOOL_TO_DWORD(StrAlg.isRuning);

(* ---- NOAlg.st ---- *)
FUNCTION_BLOCK NOAlg

VAR_IN_OUT
	StrAlg : struct_Alg;
END_VAR

VAR
	timer120 : struct_PhaseAlgoritm;
	kran6Open : struct_PhaseAlgoritm;
	pnsOn : struct_PhaseAlgoritm;
	kran4Close : struct_PhaseAlgoritm;
	kran3bOpen : struct_PhaseAlgoritm;
	mvOff : struct_PhaseAlgoritm;
	kran1Close : struct_PhaseAlgoritm;
	kran2Close : struct_PhaseAlgoritm;
	kran3Close : struct_PhaseAlgoritm;
	kran5Open : struct_PhaseAlgoritm;
	error_Krans : struct_PhaseAlgoritm;
	autoPnsOff : struct_PhaseAlgoritm;
	Pg_VhodLessThen300 : struct_PhaseAlgoritm;
	Pg_VyhodLessThen300 : struct_PhaseAlgoritm;
	nu1off : struct_PhaseAlgoritm;
	nu2off : struct_PhaseAlgoritm;
	AutoNU_Off : struct_PhaseAlgoritm;
	timer600 : struct_PhaseAlgoritm;
	pnsOff : struct_PhaseAlgoritm;
	Avom1Off : struct_PhaseAlgoritm;
	Avom2Off : struct_PhaseAlgoritm;
	Avom3Off : struct_PhaseAlgoritm;
	Avom4Off : struct_PhaseAlgoritm;
	autoAVOMOff : struct_PhaseAlgoritm;
	timer5 : struct_PhaseAlgoritm;
	klapan1 : struct_PhaseAlgoritm;
	klapan2 : struct_PhaseAlgoritm;
	nu_On : struct_PhaseAlgoritm;
	fb_timer120 : fb_ph_Timer;
	fb_kran6Open : fb_ph_Kran;
	fb_pnsOn : fb_ph_Switch;
	fb_kran4Close : fb_ph_Kran;
	fb_kran3bOpen : fb_ph_Kran;
	fb_mvOff : fb_ph_SectionSwitch;
	fb_kran1Close : fb_ph_Kran;
	fb_kran2Close : fb_ph_Kran;
	fb_kran3Close : fb_ph_Kran;
	fb_kran5Open : fb_ph_Kran;
	fb_error_Krans : fb_ph_CustomPhase;
	fb_autoPnsOff : fb_ph_algoritm;
	fb_Pg_VhodLessThen300 : fb_ph_CustomPhase;
	fb_Pg_VyhodLessThen300 : fb_ph_CustomPhase;
	fb_nu1Off : fb_ph_OilPump;
	fb_nu2Off : fb_ph_OilPump;
	fb_autoNuOff : fb_ph_algoritm;
	fb_timer600 : fb_ph_Timer;
	fb_pnsOff : fb_ph_Switch;
	fb_Avom1Off : fb_ph_Switch;
	fb_Avom2Off : fb_ph_Switch;
	fb_Avom3Off : fb_ph_Switch;
	fb_Avom4Off : fb_ph_Switch;
	fb_autoAVOMOff : fb_ph_algoritm;
	fb_timer5 : fb_ph_Timer;
	fb_klapan1 : fb_ph_CustomPhase;
	fb_klapan2 : fb_ph_CustomPhase;
	fb_nu_On : fb_ph_CustomPhase;
	_sunpackerCommand : fb_sunpackerCommand;
	_statusAi : TYPE_StatusAi;
	_Answers : TYPE_Answers;
	_statusDualInput : TYPE_statusDualInput;
	_commandDualInput : TYPE_commandDualInput;
	_DualStateImAction : TYPE_DualStateImAction;
	_PhaseAlgoritmAction : TYPE_PhaseAlgoritmAction;
	source : BYTE;
	cmd : BYTE;
	lastCmd : BYTE;
	source_for_Status : BYTE;
	cmd_for_Status : BYTE;
	command_error_for_Status : BYTE;
	resetCmdTimer : TON;
	resetCmdTimerPriznak : BOOL;
	onInit : BOOL;
	waitReset : TON;
END_VAR

VAR_EXTERNAL
	IM : ImConfig;
	algoritms : AlgoritmsConfig;
	ai : AiConfig;
	protections : ProtectionsConfig;
	ModeGpa : TYPE_ModeGpa;
	algManager : struct_AlgoritmsManager;
	AlgTimers : struct_AlgTimers;
END_VAR

VAR CONSTANT
	Ust_Pgaza : LREAL          := 0.3;
END_VAR

IF NOT onInit THEN
    fb_timer120(phaseNumber:=1, delay:=T#120S);
    fb_kran6Open(phaseNumber:=2, act:=_on);
    fb_kran4Close(phaseNumber:=3, act:=_off);
    fb_kran3bOpen(phaseNumber:=4, act:=_off);
    fb_mvOff(phaseNumber:=5, act:=_off);
    fb_kran1Close(phaseNumber:=6, act:=_off);
    fb_kran2Close(phaseNumber:=7, act:=_off);
    fb_kran3Close(phaseNumber:=8, act:=_off);
    fb_kran5Open(phaseNumber:=9, act:=_on);
    fb_error_Krans(phaseNumber:=10);
    fb_autoPnsOff(phaseNumber:=11, act:=_reset, waitCompletion:=FALSE);
    fb_pnsOn(phaseNumber:=12, act:=_on);
    fb_Pg_VhodLessThen300(phaseNumber:=13);
    fb_Pg_VyhodLessThen300(phaseNumber:=14);
    fb_nu1Off(phaseNumber:=15, act:=_off);
    fb_nu2Off(phaseNumber:=16, act:=_off);
    fb_autoNuOff(phaseNumber:=17, act:=_reset, waitCompletion:=FALSE);
    fb_timer600(phaseNumber:=18, delay:=T#600S);
    fb_pnsOff(phaseNumber:=19, act:=_off);
    fb_Avom1Off(phaseNumber:=20, act:=_off);
    fb_Avom2Off(phaseNumber:=21, act:=_off);
    fb_Avom3Off(phaseNumber:=22, act:=_off);
    fb_Avom4Off(phaseNumber:=23, act:=_off);
    fb_autoAVOMOff(phaseNumber:=24, act:=_reset, waitCompletion:=FALSE);
    fb_timer5(phaseNumber:=25, delay:=T#5S);
    fb_klapan1(phaseNumber:=26);
    fb_klapan2(phaseNumber:=27);
    fb_nu_On(phaseNumber:=28);

onInit:=TRUE;
END_IF;

fb_timer120(StrPh:=timer120, timer:=AlgTimers.No_wait120);
fb_kran6Open(StrPh:=kran6Open, Im:=Im.kran6);
fb_pnsOn(StrPh:=pnsOn, Im:=Im.pns);
fb_kran4Close(StrPh:=kran4Close, Im:=Im.kran4);
fb_kran3bOpen(StrPh:=kran3bOpen, Im:=Im.kran3b);
fb_mvOff(StrPh:=mvOff, Im:=Im.mv);
fb_kran1Close(StrPh:=kran1Close, Im:=Im.kran1);
fb_kran2Close(StrPh:=kran2Close, Im:=Im.Kran2);
fb_kran3Close(StrPh:=kran3Close, Im:=Im.Kran3);
fb_kran5Open(StrPh:=kran5Open, Im:=Im.Kran5);
fb_error_Krans(StrPh:=error_Krans);
fb_autoPnsOff(StrPh:=autoPnsOff, alg:=algoritms.autoPns);
fb_Pg_VhodLessThen300(StrPh:=Pg_VhodLessThen300);
fb_Pg_VyhodLessThen300(StrPh:=Pg_VyhodLessThen300);
fb_nu1Off(StrPh:=nu1off, Im:=Im.nu1);
fb_nu2Off(StrPh:=nu2off, Im:=Im.nu2);
fb_autoNuOff(StrPh:=AutoNU_Off, alg:=algoritms.autoNu);
fb_timer600(StrPh:=timer600, timer:=AlgTimers.No_wait600);
fb_pnsOff(StrPh:=pnsOff, Im:=Im.pns);
fb_Avom1Off(StrPh:=Avom1Off, Im:=Im.v1_Avom);
fb_Avom2Off(StrPh:=Avom2Off, Im:=Im.v2_Avom);
fb_Avom3Off(StrPh:=Avom3Off, Im:=Im.v3_Avom);
fb_Avom4Off(StrPh:=Avom4Off, Im:=Im.v4_Avom);
fb_autoAVOMOff(StrPh:=autoAVOMOff, alg:=algoritms.AutoAvom);
fb_timer5(StrPh:=timer5, timer:=AlgTimers.No_wait5);
fb_klapan1(StrPh:=klapan1);
fb_klapan2(StrPh:=klapan2);
fb_nu_On(StrPh:=nu_On);

StrAlg.CanRun := StrAlg.inCanRun;
StrAlg.OpcCommandsDisabled := StrAlg.inOpcCommandsDisabled;

IF StrAlg.isRuning THEN
    (* кран 6 не открыт - запуск таймера *)
    IF NOT kran6Open.top AND NOT timer120.top  THEN
	runPhase(timer120);
    ELSE
    (* счетчик отработал и кран 6 не открыт - ошибка *)
        IF timer120.top AND NOT kran6Open.top THEN
            error_Krans.error := TRUE;
        END_IF;
    END_IF;

    (* старт смазки кранов *)
    IF (*algoritms.F3.Smazka_1_2 OR *)IM.kran1.onStatus = _statusDualInput.STATUS_ON OR IM.kran1.onStatus = _statusDualInput.STATUS_TRANSITIONAL
	OR IM.kran2.onStatus = _statusDualInput.STATUS_ON OR IM.kran2.onStatus = _statusDualInput.STATUS_TRANSITIONAL  THEN
        IF (*(algoritms.F3.Smazka_1_2 OR *)IM.kran1.onStatus = _statusDualInput.STATUS_ON OR IM.kran1.onStatus = _statusDualInput.STATUS_TRANSITIONAL AND NOT klapan1.start AND NOT kran1Close.top THEN
            runPhase(klapan1);
        END_IF;
        IF (*(algoritms.F3.Smazka_1_2 OR *)IM.kran2.onStatus = _statusDualInput.STATUS_ON OR IM.kran2.onStatus = _statusDualInput.STATUS_TRANSITIONAL AND NOT klapan2.start AND NOT kran2Close.top THEN
            runPhase(klapan2);
        END_IF;
    (*algoritms.F3.Smazka_1_2:=FALSE;*)
    END_IF;

    (* открыть кран 6 кран 4 *)
    runPhase(kran6Open);
    runPhase(kran4Close);

    (*не понимаю
    IF kran4Close.top THEN
        ystavki.Block_kr4_alg.setValue (0);
    END_IF;*)

    (* кран 6 открыт *)
    IF kran6Open.top THEN
	runPhase(kran3bOpen);
	resetPhase(timer120);
	(*error_Krans.top := FALSE;
	error_Krans.error := FALSE;*)
	(*algoritms.S_Vibr.CanRun:=FALSE;
	algoritms.S_Vibr.reset (); net takogo alg*)
    END_IF;
    IF kran3bOpen.top AND NOT mvoff.start THEN
	resetDiProtection(protections.mvOff);
	resetDiProtection(protections.Off_avar_vikluchatel);
	resetDiProtection(protections.Reg_vozb_off);
	runPhase(mvOff);
    END_IF;

    IF mvOff.top (*AND NOT flag1*) THEN
        algoritms.AutoPns.inCanRun :=FALSE;
        (*algoritms.AutoPNS_Start.reset (); nichego ne ponimau
        algoritms.AutoPns.inCanRun :=FALSE;*)
        runPhase(autoPnsOff);
        runPhase(pnsOn);
        resetDiProtection(protections.Kran1_sdvig);
        resetDiProtection(protections.Kran2_sdvig);
        runPhase(kran1Close);
        runPhase(kran2Close);
        runPhase(kran3Close);
        runPhase(nu_On);

        (*тут запустить насосы уплотнения *)

        (*algoritms.autoNu.inCanRun:=FALSE;
        algoritms.autoNu_2.reset ();
        algoritms.autoNu_1.inCanRun:=TRUE;
        algoritms.autoNu_1.run ();
        flag1:=TRUE; что тут происходит?*)
    END_IF;
    IF ((IM.nu1.onStatus =_statusDualInput.STATUS_ON) OR (IM.nu2.onStatus =_statusDualInput.STATUS_ON)) AND nu_On.start AND NOT nu_On.top THEN
        nu_On.top:=TRUE;
    END_IF;

    (* выдача смазки *)
    IF klapan1.start AND kran1Close.top THEN
        (*IM.Kr1_Smazka.impulse(); не понимаю((((((((*)
        klapan1.top:=TRUE;
    END_IF;

    IF klapan2.start AND kran2Close.top THEN
	(*IM.Kr2_Smazka.impulse(); не понимаю *)
	klapan2.top:=TRUE;
    END_IF;

    (* кран 1 кран 2 кран 3 кран 4 закрыты - открыть кран 5 *)
    IF kran1Close.top AND kran2Close.top AND kran3Close.top AND kran4Close.top THEN
        runPhase(kran5Open);
        resetAiProtection(protections.Pgaza_na_vyhode_nagnetatelia);
    END_IF;

    IF kran5Open.top THEN
        runPhase(Pg_VhodLessThen300);
        runPhase(Pg_VyhodLessThen300);
    END_IF;

    IF Pg_VhodLessThen300.start AND NOT Pg_VhodLessThen300.top THEN
        IF (ai.Pgaza_na_vhode_nagnetatelia.interval>= _statusAi.NORMAL) AND (ai.Pgaza_na_vhode_nagnetatelia.value < 0.3) THEN
            Pg_VhodLessThen300.top:=TRUE;
        END_IF;
    END_IF;

    IF Pg_VyhodLessThen300.start AND NOT Pg_VyhodLessThen300.top THEN
        IF (ai.Pgaza_na_vyhode_nagnetatelia.interval>=_statusAi.NORMAL) AND (ai.Pgaza_na_vyhode_nagnetatelia.value < 0.3) THEN
            Pg_VyhodLessThen300.top:=TRUE;
        END_IF;
    END_IF;

    IF Pg_VhodLessThen300.top AND Pg_VyhodLessThen300.top AND pnsOn.top AND nu_On.top AND mvOff.top  THEN
        runphase(nu1Off);
        runphase(nu2Off);

        resetAiProtection(protections.dPmaslo_gaz);
        resetDiProtection(protections.dPmaslo_gaz_less100);

        runAiProtection(protections.Pgaza_na_vyhode_nagnetatelia_GPA_STOP);
        runAiProtection(protections.Pgaza_na_vhode_nagnetatelia_GPA_STOP);
        algoritms.autoNu.CanRun:=FALSE;
        AutoNU_Off.top:=TRUE;
        (*algoritms.autoNu_1.reset(); кого, чего куда*)
    END_IF;

    IF nu1Off.top THEN
        IF (*NOT algManager.reg_V AND кто чего*) NOT pnsoff.start THEN
            runPhase(timer600);
        END_IF;
        (*IF NOT pnsoff.start THEN
            sbrosVibeg.ask();
        END_IF; kto chego?*)
    END_IF;

    IF timer600.top (*OR sbrosVibeg.answer=Answers.ANS_YES kto chto *)THEN
	runPhase(pnsOff);
	resetAiProtection(protections.Pmaslo_sm_nizkoe);
	resetAiProtection(protections.Pmaslo_sm_vysokoe);
	(*sbrosVibeg.reset (); pomogite *)
	resetPhase(timer600);
	(*algoritms.F2_Ch.autoAVOM_canrun_flag:=FALSE;
	algoritms.F2_R.autoAVOM_canrun_flag:=FALSE;*)
    END_IF;
    IF (*(NOT algoritms.F2_Ch.autoAVOM_canrun_flag) AND (NOT algoritms.F2_R.autoAVOM_canrun_flag) AND*)pnsoff.start THEN
	runPhase(Avom1Off);
	runPhase(Avom2Off);
	runPhase(Avom3Off);
	runPhase(Avom4Off);

	(*algoritms.R_AutoAVOM.CanRun:=FALSE;
	algoritms.R_AutoAVOM.reset();
	algoritms.S_AutoAVOM.CanRun:=FALSE;
	algoritms.S_AutoAVOM.reset();
	algoritms.Auto_Avom_.CanRun:=FALSE;*)
	runPhase(autoAVOMOff);
    END_IF;

    IF pnsOff.top AND Avom1Off.top AND Avom2Off.top AND Avom3Off.top AND Avom4Off.top AND autoAVOMOff.top  THEN
        runPhase(timer5);
    END_IF;

    IF timer5.top THEN
	resetPhase(timer5);
    END_IF;
END_IF;

_sunpackerCommand(command := StrAlg.inCommand);
	source := _sunpackerCommand.source;
	cmd := _sunpackerCommand.cmd;

IF cmd <> 0 AND lastCmd <> cmd AND (((NOT StrAlg.opcCommandsDisabled) AND source > 0) OR source = 0) then
	CASE BYTE_TO_INT(cmd) OF
		(*cmdRun*) 1: 	IF (StrAlg.CanRun) THEN
					StrAlg.isRuning := TRUE;
					StrAlg.isEnded := FALSE;
					StrAlg.hasError := FALSE;
					(*****************       OnRun       *****************)

                                                  algManager.nMode:=ModeGpa.MODE_NO;
                                                  (*runIfNotRunningSO(IM.SingleOutputs.Lampa_NO);*)

                                                  runPhase(kran4Close);
                                                  runPhase(timer120);
                                                  runPhase(nu1Off);
                                                  runPhase(timer600);

                                                 (* resetAiProtection(protections.Pgaza_na_vyhode_nagnetatelia);
                                                  resetAiProtection(protections.dPmaslo_gaz);
                                                  resetAiProtection(protections.Pmaslo_sm_nizkoe);
                                                  resetAiProtection(protections.Pmaslo_sm_vysokoe);
                                                  resetAiProtection(protections.Pgaza_na_vhode_nagnetatelia);
                                                  resetAiProtection(protections.Pgaza_na_vyhode_nagnetatelia);
                                                  resetDiProtection(protections.Reg_vozb_off);
                                                  resetDiProtection(protections.Fail_chastotnii_pusk);*)

					cmd_for_Status := cmd;
					source_for_Status := source;
					command_error_for_Status := 0;
				ELSE
					StrAlg.isRuning := FALSE;
					StrAlg.isEnded := FALSE;
					StrAlg.hasError 	:= FALSE;

					cmd_for_Status := 0;
					source_for_Status := source;
					command_error_for_Status := cmd;
				END_IF;
		(*cmdReset*) 2: 	StrAlg.isRuning := FALSE;
				StrAlg.isEnded := FALSE;
				StrAlg.hasError 	:= FALSE;

                                         (*****************       OnReset       *****************)
                                        waitReset(IN:=FALSE);
                                        (*resetIfRunningSO(IM.SingleOutputs.Lampa_NO);*)
                                        resetIfRunning(algoritms.vibegPNS);
                                        (*impulseSO(Im.SingleOutputs.SbrosBREO);*)

                                        resetPhase(timer120);
                                        resetPhase(kran6Open);
                                        resetPhase(pnsOn);
                                        resetPhase(kran4Close);
                                        resetPhase(kran3bOpen);
                                        resetPhase(mvOff);
                                        resetPhase(kran1Close);
                                        resetPhase(kran2Close);
                                        resetPhase(kran3Close);
                                        resetPhase(kran5Open);
	                              resetPhase(error_Krans);
                                        resetPhase(autoPnsOff);
                                        resetPhase(pnsOn);
                                        resetPhase(Pg_VhodLessThen300);
                                        resetPhase(Pg_VyhodLessThen300);
                                        resetPhase(nu2Off);
                                        resetPhase(nu1Off);
                                        resetPhase(AutoNU_Off);
                                        resetPhase(timer600);

				cmd_for_Status := cmd;
				source_for_Status := source;
				command_error_for_Status := 0;
	END_CASE;
	resetCmdTimer(IN := false);
	resetCmdTimerPriznak := TRUE;
END_IF;
lastCmd := cmd;

resetCmdTimer(IN := resetCmdTimerPriznak, PT := T#5S);
IF resetCmdTimer.Q THEN
	resetCmdTimerPriznak := FALSE;
	source_for_Status := 0;
	cmd_for_Status := 0;
	command_error_for_Status := 0;
END_IF;

StrAlg.Start:= timer120.startStatus
            OR kran6Open.startStatus
            OR pnsOn.startStatus
            OR kran4Close.startStatus
            OR kran3bOpen.startStatus
            OR mvOff.startStatus
            OR kran1Close.startStatus
            OR kran2Close.startStatus
            OR kran3Close.startStatus
            OR kran5Open.startStatus
            OR error_Krans.startStatus
            OR autoPnsOff.startStatus
            OR pnsOn.startStatus
            OR Pg_VhodLessThen300.startStatus
            OR Pg_VyhodLessThen300.startStatus
            OR nu2Off.startStatus
            OR nu1Off.startStatus
            OR AutoNU_Off.startStatus
            OR timer600.startStatus;

StrAlg.Error:= timer120.errorStatus
            OR kran6Open.errorStatus
            OR pnsOn.errorStatus
            OR kran4Close.errorStatus
            OR kran3bOpen.errorStatus
            OR mvOff.errorStatus
            OR kran1Close.errorStatus
            OR kran2Close.errorStatus
            OR kran3Close.errorStatus
            OR kran5Open.errorStatus
            OR error_Krans.errorStatus
            OR autoPnsOff.errorStatus
            OR pnsOn.errorStatus
            OR Pg_VhodLessThen300.errorStatus
            OR Pg_VyhodLessThen300.errorStatus
            OR nu2Off.errorStatus
            OR nu1Off.errorStatus
            OR AutoNU_Off.errorStatus
            OR timer600.errorStatus;

StrAlg.Top:=   timer120.topStatus
            OR kran6Open.topStatus
            OR pnsOn.topStatus
            OR kran4Close.topStatus
            OR kran3bOpen.topStatus
            OR mvOff.topStatus
            OR kran1Close.topStatus
            OR kran2Close.topStatus
            OR kran3Close.topStatus
            OR kran5Open.topStatus
            OR error_Krans.topStatus
            OR autoPnsOff.topStatus
            OR pnsOn.topStatus
            OR Pg_VhodLessThen300.topStatus
            OR Pg_VyhodLessThen300.topStatus
            OR nu2Off.topStatus
            OR nu1Off.topStatus
            OR AutoNU_Off.topStatus
            OR timer600.topStatus;

(*TODO: TYPE PROGRAM CODE HERE*)
StrAlg.status :=  SHL(BYTE_TO_DWORD(source_for_Status), 29)
			OR SHL(BYTE_TO_DWORD(cmd_for_Status), 26)
			OR SHL(BYTE_TO_DWORD(command_error_for_Status), 23)
			OR SHL(BOOL_TO_DWORD(StrAlg.OpcCommandsDisabled ), 21)
			OR SHL(BOOL_TO_DWORD(StrAlg.hasError),4)
			OR SHL(BOOL_TO_DWORD(StrAlg.CanRun),2)
			OR SHL(BOOL_TO_DWORD(StrAlg.isEnded),1)
			OR BOOL_TO_DWORD(StrAlg.isRuning);
